(* CODESYS project OPAK_RFID.LIBRARY
   DefaultNamespace: ELA_OPAK_RFID
   Author: elrest Automationssysteme GmbH
   Title: OPAK_RFID
   DocFormat: reStructuredText
   Version: 3.5.0.0
   Description: Library to acces the RFID reader/writer on the EMC500 HW
   LanguageModelAttribute: qualified-access-only
   Company: elrest Automationssysteme GmbH

Project tree, tasks and I/O mapping:
  libraries: CAA Types Extern, * (CAA Technical Workgroup); CAA Behaviour Model, * (CAA Technical Workgroup); CAA FB Factory, * (CAA Technical Workgroup)
  00000000-0000-0000-0000-000000000000|D:\CoDeSys\LibrariesV3\trunk\Intern\CAA\CAA Template\3.2.0.3 draft\Prefix.pdf
  00000000-0000-0000-0000-000000000000|D:\CoDeSys\LibrariesV3\trunk\Intern\CAA\CAA Template\3.4.0.0 draft\Placeholder.xml
  00000000-0000-0000-0000-000000000000|D:\CoDeSys\LibrariesV3\trunk\Intern\CAA\CAA Template\3.5.2.0 draft\Placeholder.xml
  Libname/
    Enums/
      data type ERROR
    Function Blocks/
    Functions/
      function isTagPresent [ST]
      function getTagID [ST]
      function readFromTag [ST]
      function writeToTag [ST]
    GlobalConstants/
      global variables Constants
    GlobalVariables/
      global variables Variables
    Interfaces/
    Structs/
    Templates/
      Behaviour Model/
        function block ETrigA_Temp [ST]: prvAbort, prvCyclicAction, prvResetOutputs, prvStart
        function block ETrigTlA_Temp [ST]: prvAbort, prvCyclicAction, prvResetOutputs, prvStart
        function block ETrigTl_Temp [ST]: prvAbort, prvCyclicAction, prvResetOutputs, prvStart
        function block ETrigToA_Temp [ST]: prvAbort, prvCyclicAction, prvResetOutputs, prvStart
        function block ETrigToTlA_Temp [ST]: prvAbort, prvCyclicAction, prvResetOutputs, prvStart
        function block ETrigToTl_Temp [ST]: prvAbort, prvCyclicAction, prvResetOutputs, prvStart
        function block ETrigTo_Temp [ST]: prvAbort, prvCyclicAction, prvResetOutputs, prvStart
        function block ETrig_Temp [ST]: prvAbort, prvCyclicAction, prvResetOutputs, prvStart
        function block LTrig_Temp [ST]: prvAbort, prvCyclicAction, prvResetOutputs, prvStart
      FB Factory/
        function block CustomData [ST]
        function block CustomFB [ST]: prvInstInit
        function block CustomFBFactory_heap [ST]: Create, prvInstCount, prvInstPoolExtendsFactor, prvInstSize
        function block CustomFBFactory_static [ST]: Create, prvInstPoolAdr, prvInstPoolSize, prvInstSize
    Types/
  Projektinformationen/
    function GetCompany [ST]
    function GetTitle [ST]
    function GetVersion [ST]
    function GetTextProperty [ST]
    function GetNumberProperty [ST]
    function GetBooleanProperty [ST]
    function GetVersionProperty [ST]
*)

// Libname/Enums/ERROR
{attribute 'qualified_only'}
//{attribute 'conditionalshow'}
//{attribute 'conditionalshow' := 'SomeText'}
//{attribute 'hide'}
TYPE ERROR : (NO_ERROR, TIME_OUT); END_TYPE

// Libname/GlobalConstants/Constants
{attribute 'qualified_only'}
//{attribute 'conditionalshow'}
//{attribute 'conditionalshow' := 'SomeText'}
//{attribute 'hide'}
VAR_GLOBAL CONSTANT
	gc_iDummy : INT := 42; /// This is a dummy global constant variable
END_VAR

// Libname/GlobalVariables/Variables
{attribute 'qualified_only'}
//{attribute 'conditionalshow'}
//{attribute 'conditionalshow' := 'SomeText'}
//{attribute 'hide'}
VAR_GLOBAL
	g_iDummy : INT; /// This is a dummy global variable
END_VAR

// Libname/Templates/Behaviour Model/ETrigA_Temp
//{attribute 'hide_all_locals'}
//{attribute 'conditionalshow_all_locals' := 'SomeText'}
//{attribute 'conditionalshow_all_locals'}
//{attribute 'conditionalshow' := 'SomeText'}
//{attribute 'conditionalshow'}
//{attribute 'hide'}
FUNCTION_BLOCK ETrigA_Temp EXTENDS CBM.ETrigA
VAR_INPUT
	(* specific Inputs *)
END_VAR
VAR_OUTPUT
	eError : ERROR;
	(* specific Outputs *)
END_VAR
VAR
	(* specific vars *)
END_VAR

SUPER^();
IF iError = CBM.ERROR.TIME_OUT THEN
	eError := ERROR.TIME_OUT;
ELSE
	eError := iError;
END_IF

{attribute 'hide'}
METHOD prvAbort : BOOL
VAR_INPUT
END_VAR
VAR
END_VAR
IF xError THEN (* abort because of error *)
	(* TODO: insert specific Code here *)
ELSE (* user abort *)
	(* TODO: insert specific Code here *)
END_IF
xAbortInProgress:= FALSE;
END_METHOD

{attribute 'hide'}
METHOD prvCyclicAction : BOOL
VAR_INPUT
END_VAR
VAR
END_VAR
(* TODO: insert specific Code here *)
xDone:= TRUE;
(* if an error occurs, set iError to a value else than zero instead of xDone:= TRUE *)
(* to keep repeat loop *)
END_METHOD

{attribute 'hide'}
METHOD prvResetOutputs : BOOL
VAR_INPUT
END_VAR
VAR
END_VAR
(* TODO: insert specific Code here *)
SUPER^.prvResetOutputs();
END_METHOD

{attribute 'hide'}
METHOD prvStart : BOOL
VAR_INPUT
END_VAR
VAR
END_VAR
(* this code is called, when the application is started (rising edge of xExecute *)
(* TODO: copy specific input variables into local copies *)
(* TODO: insert specific Code here *)
;
END_METHOD

END_FUNCTION_BLOCK

// Libname/Templates/Behaviour Model/ETrigTlA_Temp
//{attribute 'hide_all_locals'}
//{attribute 'conditionalshow_all_locals' := 'SomeText'}
//{attribute 'conditionalshow_all_locals'}
//{attribute 'conditionalshow' := 'SomeText'}
//{attribute 'conditionalshow'}
//{attribute 'hide'}
FUNCTION_BLOCK ETrigTlA_Temp EXTENDS CBM.ETrigTlA
VAR_INPUT
	(* specific Inputs *)
END_VAR
VAR_OUTPUT
	eError : ERROR;
	(* specific Outputs *)
END_VAR
VAR
	(* specific vars *)
END_VAR

SUPER^();
IF iError = CBM.ERROR.TIME_OUT THEN
	eError := ERROR.TIME_OUT;
ELSE
	eError := iError;
END_IF

{attribute 'hide'}
METHOD prvAbort : BOOL
VAR_INPUT
END_VAR
VAR
END_VAR
IF xError THEN (* abort because of error *)
	(* TODO: insert specific Code here *)
ELSE (* user abort *)
	(* TODO: insert specific Code here *)
END_IF
xAbortInProgress:= FALSE;
END_METHOD

{attribute 'hide'}
METHOD prvCyclicAction : BOOL
VAR_INPUT
END_VAR
VAR
END_VAR
(* TODO: insert specific Code here *)
xDone:= TRUE;
(* if an error occurs, set iError to a value else than zero instead of xDone:= TRUE *)
(* to keep repeat loop *)
END_METHOD

{attribute 'hide'}
METHOD prvResetOutputs : BOOL
VAR_INPUT
END_VAR
VAR
END_VAR
(* TODO: insert specific Code here *)
SUPER^.prvResetOutputs();
END_METHOD

{attribute 'hide'}
METHOD prvStart : BOOL
VAR_INPUT
END_VAR
VAR
END_VAR
(* this code is called, when the application is started (rising edge of xExecute *)
(* TODO: copy specific input variables into local copies *)
(* TODO: insert specific Code here *)
;
END_METHOD

END_FUNCTION_BLOCK

// Libname/Templates/Behaviour Model/ETrigTl_Temp
//{attribute 'hide_all_locals'}
//{attribute 'conditionalshow_all_locals' := 'SomeText'}
//{attribute 'conditionalshow_all_locals'}
//{attribute 'conditionalshow' := 'SomeText'}
//{attribute 'conditionalshow'}
//{attribute 'hide'}
FUNCTION_BLOCK ETrigA_Temp EXTENDS CBM.ETrigTl
VAR_INPUT
	(* specific Inputs *)
END_VAR
VAR_OUTPUT
	eError : ERROR;
	(* specific Outputs *)
END_VAR
VAR
	(* specific vars *)
END_VAR

SUPER^();
IF iError = CBM.ERROR.TIME_OUT THEN
	eError := ERROR.TIME_OUT;
ELSE
	eError := iError;
END_IF

{attribute 'hide'}
METHOD prvAbort : BOOL
VAR_INPUT
END_VAR
VAR
END_VAR
IF xError THEN (* abort because of error *)
	(* TODO: insert specific Code here *)
ELSE (* user abort *)
	(* TODO: insert specific Code here *)
END_IF
xAbortInProgress:= FALSE;
END_METHOD

{attribute 'hide'}
METHOD prvCyclicAction : BOOL
VAR_INPUT
END_VAR
VAR
END_VAR
(* TODO: insert specific Code here *)
xDone:= TRUE;
(* if an error occurs, set iError to a value else than zero instead of xDone:= TRUE *)
(* to keep repeat loop *)
END_METHOD

{attribute 'hide'}
METHOD prvResetOutputs : BOOL
VAR_INPUT
END_VAR
VAR
END_VAR
(* TODO: insert specific Code here *)
SUPER^.prvResetOutputs();
END_METHOD

{attribute 'hide'}
METHOD prvStart : BOOL
VAR_INPUT
END_VAR
VAR
END_VAR
(* this code is called, when the application is started (rising edge of xExecute *)
(* TODO: copy specific input variables into local copies *)
(* TODO: insert specific Code here *)
;
END_METHOD

END_FUNCTION_BLOCK

// Libname/Templates/Behaviour Model/ETrigToA_Temp
//{attribute 'hide_all_locals'}
//{attribute 'conditionalshow_all_locals' := 'SomeText'}
//{attribute 'conditionalshow_all_locals'}
//{attribute 'conditionalshow' := 'SomeText'}
//{attribute 'conditionalshow'}
//{attribute 'hide'}
FUNCTION_BLOCK ETrigToA_Temp EXTENDS CBM.ETrigToA
VAR_INPUT
	(* specific Inputs *)
END_VAR
VAR_OUTPUT
	eError : ERROR;
	(* specific Outputs *)
END_VAR
VAR
	(* specific vars *)
END_VAR

SUPER^();
IF iError = CBM.ERROR.TIME_OUT THEN
	eError := ERROR.TIME_OUT;
ELSE
	eError := iError;
END_IF

{attribute 'hide'}
METHOD prvAbort : BOOL
VAR_INPUT
END_VAR
VAR
END_VAR
IF xError THEN (* abort because of error *)
	(* TODO: insert specific Code here *)
ELSE (* user abort *)
	(* TODO: insert specific Code here *)
END_IF
xAbortInProgress:= FALSE;
END_METHOD

{attribute 'hide'}
METHOD prvCyclicAction : BOOL
VAR_INPUT
END_VAR
VAR
END_VAR
(* TODO: insert specific Code here *)
xDone:= TRUE;
(* if an error occurs, set iError to a value else than zero instead of xDone:= TRUE *)
END_METHOD

{attribute 'hide'}
METHOD prvResetOutputs : BOOL
VAR_INPUT
END_VAR
VAR
END_VAR
(* TODO: insert specific Code here *)
SUPER^.prvResetOutputs();
END_METHOD

{attribute 'hide'}
METHOD prvStart : BOOL
VAR_INPUT
END_VAR
VAR
END_VAR
(* this code is called, when the application is started (rising edge of xExecute *)
(* TODO: copy specific input variables into local copies *)
(* TODO: insert specific Code here *)
;
END_METHOD

END_FUNCTION_BLOCK

// Libname/Templates/Behaviour Model/ETrigToTlA_Temp
//{attribute 'hide_all_locals'}
//{attribute 'conditionalshow_all_locals' := 'SomeText'}
//{attribute 'conditionalshow_all_locals'}
//{attribute 'conditionalshow' := 'SomeText'}
//{attribute 'conditionalshow'}
//{attribute 'hide'}
FUNCTION_BLOCK ETrigToTlA_Temp EXTENDS CBM.ETrigToTlA
VAR_INPUT
	(* specific Inputs *)
END_VAR
VAR_OUTPUT
	eError : ERROR;
	(* specific Outputs *)
END_VAR
VAR
	(* specific vars *)
END_VAR

SUPER^();
IF iError = CBM.ERROR.TIME_OUT THEN
	eError := ERROR.TIME_OUT;
ELSE
	eError := iError;
END_IF

{attribute 'hide'}
METHOD prvAbort : BOOL
VAR_INPUT
END_VAR
VAR
END_VAR
IF xError THEN (* abort because of error *)
	(* TODO: insert specific Code here *)
ELSE (* user abort *)
	(* TODO: insert specific Code here *)
END_IF
xAbortInProgress:= FALSE;
END_METHOD

{attribute 'hide'}
METHOD prvCyclicAction : BOOL
VAR_INPUT
END_VAR
VAR
END_VAR
(* TODO: insert specific Code here *)
xDone:= TRUE;
(* if an error occurs, set iError to a value else than zero instead of xDone:= TRUE *)
(* to keep repeat loop *)
END_METHOD

{attribute 'hide'}
METHOD prvResetOutputs : BOOL
VAR_INPUT
END_VAR
VAR
END_VAR
(* TODO: insert specific Code here *)
SUPER^.prvResetOutputs();
END_METHOD

{attribute 'hide'}
METHOD prvStart : BOOL
VAR_INPUT
END_VAR
VAR
END_VAR
(* this code is called, when the application is started (rising edge of xExecute *)
(* TODO: copy specific input variables into local copies *)
(* TODO: insert specific Code here *)
;
END_METHOD

END_FUNCTION_BLOCK

// Libname/Templates/Behaviour Model/ETrigToTl_Temp
//{attribute 'hide_all_locals'}
//{attribute 'conditionalshow_all_locals' := 'SomeText'}
//{attribute 'conditionalshow_all_locals'}
//{attribute 'conditionalshow' := 'SomeText'}
//{attribute 'conditionalshow'}
//{attribute 'hide'}
FUNCTION_BLOCK ETrigToTl_Temp EXTENDS CBM.ETrigToTl
VAR_INPUT
	(* specific Inputs *)
END_VAR
VAR_OUTPUT
	eError : ERROR;
	(* specific Outputs *)
END_VAR
VAR
	(* specific vars *)
END_VAR

SUPER^();
IF iError = CBM.ERROR.TIME_OUT THEN
	eError := ERROR.TIME_OUT;
ELSE
	eError := iError;
END_IF

{attribute 'hide'}
METHOD prvAbort : BOOL
VAR_INPUT
END_VAR
VAR
END_VAR
IF xError THEN (* abort because of error *)
	(* TODO: insert specific Code here *)
ELSE (* user abort *)
	(* TODO: insert specific Code here *)
END_IF
xAbortInProgress:= FALSE;
END_METHOD

{attribute 'hide'}
METHOD prvCyclicAction : BOOL
VAR_INPUT
END_VAR
VAR
END_VAR
(* TODO: insert specific Code here *)
xDone:= TRUE;
(* if an error occurs, set iError to a value else than zero instead of xDone:= TRUE *)
(* to keep repeat loop *)
END_METHOD

{attribute 'hide'}
METHOD prvResetOutputs : BOOL
VAR_INPUT
END_VAR
VAR
END_VAR
(* TODO: insert specific Code here *)
SUPER^.prvResetOutputs();
END_METHOD

{attribute 'hide'}
METHOD prvStart : BOOL
VAR_INPUT
END_VAR
VAR
END_VAR
(* this code is called, when the application is started (rising edge of xExecute *)
(* TODO: copy specific input variables into local copies *)
(* TODO: insert specific Code here *)
;
END_METHOD

END_FUNCTION_BLOCK

// Libname/Templates/Behaviour Model/ETrigTo_Temp
//{attribute 'hide_all_locals'}
//{attribute 'conditionalshow_all_locals' := 'SomeText'}
//{attribute 'conditionalshow_all_locals'}
//{attribute 'conditionalshow' := 'SomeText'}
//{attribute 'conditionalshow'}
//{attribute 'hide'}
FUNCTION_BLOCK ETrigTo_Temp EXTENDS CBM.ETrigTo
VAR_INPUT
	(* specific Inputs *)
END_VAR
VAR_OUTPUT
	eError : ERROR;
	(* specific Outputs *)
END_VAR
VAR
	(* specific vars *)
END_VAR

SUPER^();
IF iError = CBM.ERROR.TIME_OUT THEN
	eError := ERROR.TIME_OUT;
ELSE
	eError := iError;
END_IF

{attribute 'hide'}
METHOD prvAbort : BOOL
VAR_INPUT
END_VAR
VAR
END_VAR
IF xError THEN (* abort because of error *)
	(* TODO: insert specific Code here *)
ELSE (* user abort *)
	(* TODO: insert specific Code here *)
END_IF
xAbortInProgress:= FALSE;
END_METHOD

{attribute 'hide'}
METHOD prvCyclicAction : BOOL
VAR_INPUT
END_VAR
VAR
END_VAR
(* TODO: insert specific Code here *)
xDone:= TRUE;
(* if an error occurs, set iError to a value else than zero instead of xDone:= TRUE *)
(* to keep repeat loop *)
END_METHOD

{attribute 'hide'}
METHOD prvResetOutputs : BOOL
VAR_INPUT
END_VAR
VAR
END_VAR
(* TODO: insert specific Code here *)
SUPER^.prvResetOutputs();
END_METHOD

{attribute 'hide'}
METHOD prvStart : BOOL
VAR_INPUT
END_VAR
VAR
END_VAR
(* this code is called, when the application is started (rising edge of xExecute *)
(* TODO: copy specific input variables into local copies *)
(* TODO: insert specific Code here *)
;
END_METHOD

END_FUNCTION_BLOCK

// Libname/Templates/Behaviour Model/ETrig_Temp
//{attribute 'hide_all_locals'}
//{attribute 'conditionalshow_all_locals' := 'SomeText'}
//{attribute 'conditionalshow_all_locals'}
//{attribute 'conditionalshow' := 'SomeText'}
//{attribute 'conditionalshow'}
//{attribute 'hide'}
FUNCTION_BLOCK ETrig_Temp EXTENDS CBM.ETrig
VAR_INPUT
	(* specific Inputs *)
END_VAR
VAR_OUTPUT
	eError : ERROR;
	(* specific Outputs *)
END_VAR
VAR
	(* specific vars *)
END_VAR

SUPER^();
IF iError = CBM.ERROR.TIME_OUT THEN
	eError := ERROR.TIME_OUT;
ELSE
	eError := iError;
END_IF

{attribute 'hide'}
METHOD prvAbort : BOOL
VAR_INPUT
END_VAR
VAR
END_VAR
IF xError THEN (* abort because of error *)
	(* TODO: insert specific Code here *)
ELSE (* user abort *)
	(* TODO: insert specific Code here *)
END_IF
xAbortInProgress:= FALSE;
END_METHOD

{attribute 'hide'}
METHOD prvCyclicAction : BOOL
VAR_INPUT
END_VAR
VAR
END_VAR
(* TODO: insert specific Code here *)
xDone:= TRUE;
(* if an error occurs, set iError to a value else than zero instead of xDone:= TRUE *)
(* to keep repeat loop *)
END_METHOD

{attribute 'hide'}
METHOD prvResetOutputs : BOOL
VAR_INPUT
END_VAR
VAR
END_VAR
(* TODO: insert specific Code here *)
SUPER^.prvResetOutputs();
END_METHOD

{attribute 'hide'}
METHOD prvStart : BOOL
VAR_INPUT
END_VAR
VAR
END_VAR
(* this code is called, when the application is started (rising edge of xExecute *)
(* TODO: copy specific input variables into local copies *)
(* TODO: insert specific Code here *)
;
END_METHOD

END_FUNCTION_BLOCK

// Libname/Templates/Behaviour Model/LTrig_Temp
//{attribute 'hide_all_locals'}
//{attribute 'conditionalshow_all_locals' := 'SomeText'}
//{attribute 'conditionalshow_all_locals'}
//{attribute 'conditionalshow' := 'SomeText'}
//{attribute 'conditionalshow'}
//{attribute 'hide'}
FUNCTION_BLOCK LTrig_Temp EXTENDS CBM.LTrig
VAR_INPUT
	(* specific Inputs *)
END_VAR
VAR_OUTPUT
	eError : ERROR;
	(* specific Outputs *)
END_VAR
VAR
	(* specific vars *)
END_VAR

SUPER^();
IF iError = CBM.ERROR.TIME_OUT THEN
	eError := ERROR.TIME_OUT;
ELSE
	eError := iError;
END_IF

{attribute 'hide'}
METHOD prvAbort : BOOL
VAR_INPUT
END_VAR
VAR
END_VAR
IF xError THEN (* abort because of error *)
	(* TODO: insert specific Code here *)
ELSE (* user abort *)
	(* TODO: insert specific Code here *)
END_IF
xAbortInProgress:= FALSE;
END_METHOD

{attribute 'hide'}
METHOD prvCyclicAction : BOOL
VAR_INPUT
END_VAR
VAR
END_VAR
(* TODO: insert specific Code here *)
xDone:= TRUE;
(* if an error occurs, set iError to a value else than zero instead of xDone:= TRUE *)
(* to keep repeat loop *)
END_METHOD

{attribute 'hide'}
METHOD prvResetOutputs : BOOL
VAR_INPUT
END_VAR
VAR
END_VAR
(* TODO: insert specific Code here *)
SUPER^.prvResetOutputs();
END_METHOD

{attribute 'hide'}
METHOD prvStart : BOOL
VAR_INPUT
END_VAR
VAR
END_VAR
(* this code is called, when the application is started (rising edge of xExecute *)
(* TODO: copy specific input variables into local copies *)
(* TODO: insert specific Code here *)
;
END_METHOD

END_FUNCTION_BLOCK

// Libname/Templates/FB Factory/CustomData
// This is a container to carry init data from the Create methode of the factory
// to the prvInstInit methode of the new generated function block instance
{attribute 'enable_dynamic_creation'}
//{attribute 'hide_all_locals'}
//{attribute 'conditionalshow_all_locals' := 'SomeText'}
//{attribute 'conditionalshow_all_locals'}
//{attribute 'conditionalshow' := 'SomeText'}
//{attribute 'conditionalshow'}
//{attribute 'hide'}
FUNCTION_BLOCK CustomData EXTENDS FBF.InstanceData
VAR_INPUT
	(* Todo: Add your application specific data as input variables *)
END_VAR

(* !! Do not add any executable code here !! *)
SUPER^();

END_FUNCTION_BLOCK

// Libname/Templates/FB Factory/CustomFB
{attribute 'enable_dynamic_creation'}
//{attribute 'hide_all_locals'}
//{attribute 'conditionalshow_all_locals' := 'SomeText'}
//{attribute 'conditionalshow_all_locals'}
//{attribute 'conditionalshow' := 'SomeText'}
//{attribute 'conditionalshow'}
//{attribute 'hide'}
FUNCTION_BLOCK CustomFB EXTENDS FBF.InstanceBase;
VAR_INPUT
END_VAR
VAR_OUTPUT
END_VAR
VAR
END_VAR

SUPER^();

// This methode is called from the factory to give a chance
// to initialize the new fb instance with the content of itfData
//{attribute 'hide_all_locals'}
//{attribute 'conditionalshow_all_locals' := 'SomeText'}
//{attribute 'conditionalshow_all_locals'}
//{attribute 'conditionalshow' := 'SomeText'}
//{attribute 'conditionalshow'}
//{attribute 'hide'}
METHOD prvInstInit : FBF.ERROR
VAR_INPUT
	itfData : IData; 
END_VAR
VAR
	pData : POINTER TO CustomData;
	xOk : BOOL;
END_VAR
SUPER^.prvInstInit(itfData);
xOk := __QUERYPOINTER(itfData, pData);
IF xOk THEN
	(* THIS^.iLocalVar := pData^.iInitValue *);
END_IF
END_METHOD

END_FUNCTION_BLOCK

// Libname/Templates/FB Factory/CustomFBFactory_heap
// This is a template for a factory with an heap based extendable memory pool
{attribute 'enable_dynamic_creation'}
//{attribute 'hide_all_locals'}
//{attribute 'conditionalshow_all_locals' := 'SomeText'}
//{attribute 'conditionalshow_all_locals'}
//{attribute 'conditionalshow' := 'SomeText'}
//{attribute 'conditionalshow'}
//{attribute 'hide'}
FUNCTION_BLOCK CustomFBFactory_heap EXTENDS FactoryBase
VAR
END_VAR

SUPER^();

(* Please replace CustonFB with your specific function block type *)
(* There is no need to change anything else !!! *)
METHOD Create : POINTER TO CustomFB
VAR_INPUT
	itfData : FBF.IData;
END_VAR
VAR_OUTPUT
	eError : FBF.ERROR;
END_VAR
VAR
	hInst : CAA.HANDLE;
	itfInst : FBF.IInstance;
	xOk : BOOL;
END_VAR
(* !!! This code must not be subject to change !!! *)
hInst := SUPER^.prvAllocInstMem(eError => eError);
Create := SUPER^.prvGetInstPointer(hInst);
IF Create <> 0 AND eError = FBF.ERROR.NO_ERROR THEN

	{implicit on}
	Create^.__vfInit();
	Create^.FB_Init(TRUE, FALSE);
	{implicit off}

	xOk := __QUERYINTERFACE(Create^, itfInst);
	IF xOk THEN
		xOk := SUPER^.prvInstInit(itfInst, hInst, itfData, eError=>eError);
	ELSE
		eError := FBF.ERROR.WRONG_INTERFACE;
	END_IF

	IF NOT xOk THEN
		SUPER^.prvFreeInstMem(hInst);
		Create := CAA.gc_pNULL;
	END_IF
END_IF
END_METHOD

//{attribute 'conditionalshow' := 'SomeText'}
//{attribute 'conditionalshow'}
//{attribute 'hide'}
PROPERTY prvInstCount : CAA.COUNT (* ctInst *)
GET
(* Please choose a proper value for prvInstCount *)
prvInstCount := 10;
END_GET
END_PROPERTY

//{attribute 'conditionalshow' := 'SomeText'}
//{attribute 'conditionalshow'}
//{attribute 'hide'}
PROPERTY prvInstPoolExtendsFactor : USINT (* usiFactor [0..x%] *)
GET
(* Please choose a proper value for prvInstPoolExtendsFactor *)
(* This value will be interpreted as a 0..x% size extendsion related to the original size of the pool *)
prvInstPoolExtendsFactor := 20;
END_GET
END_PROPERTY

//{attribute 'conditionalshow' := 'SomeText'}
//{attribute 'conditionalshow'}
//{attribute 'hide'}
PROPERTY prvInstSize : CAA.SIZE (* szInst *)
GET
(* Please replace CustomFB with your specific function block type *)
prvInstSize := sizeof(CustomFB);
END_GET
END_PROPERTY

END_FUNCTION_BLOCK

// Libname/Templates/FB Factory/CustomFBFactory_static
// This is a template for a factory with an static iec memory based memory pool which a fixed capacity
{attribute 'enable_dynamic_creation'}
//{attribute 'hide_all_locals'}
//{attribute 'conditionalshow_all_locals' := 'SomeText'}
//{attribute 'conditionalshow_all_locals'}
//{attribute 'conditionalshow' := 'SomeText'}
//{attribute 'conditionalshow'}
//{attribute 'hide'}
FUNCTION_BLOCK CustomFBFactory_static EXTENDS FactoryBase
VAR
	// Please change the size of abyPoolMemory with your specific application need
	abyPoolMemory : ARRAY[0..529] OF BYTE;
END_VAR

SUPER^();

(* Please replace CustonFB with our specific function block type *)
(* There is no need to change anything else !!! *)
METHOD Create : POINTER TO CustomFB
VAR_INPUT
	itfData : FBF.IData;
END_VAR
VAR_OUTPUT
	eError : FBF.ERROR;
END_VAR
VAR
	hInst : CAA.HANDLE;
	itfInst : FBF.IInstance;
	xOk : BOOL;
END_VAR
(* !!! This code must not be subject to change !!! *)
hInst := SUPER^.prvAllocInstMem(eError => eError);
Create := SUPER^.prvGetInstPointer(hInst);
IF Create <> 0 AND eError = FBF.ERROR.NO_ERROR THEN

	{implicit on}
	Create^.__vfInit();
	Create^.FB_Init(TRUE, FALSE);
	{implicit off}

	xOk := __QUERYINTERFACE(Create^, itfInst);
	IF xOk THEN
		xOk := SUPER^.prvInstInit(itfInst, hInst, itfData, eError=>eError);
	ELSE
		eError := FBF.ERROR.WRONG_INTERFACE;
	END_IF

	IF NOT xOk THEN
		SUPER^.prvFreeInstMem(hInst);
		Create := CAA.gc_pNULL;
	END_IF
END_IF
END_METHOD

//{attribute 'conditionalshow' := 'SomeText'}
//{attribute 'conditionalshow'}
//{attribute 'hide'}
PROPERTY prvInstPoolAdr : CAA.PVOID (* pPool *)
GET
prvInstPoolAdr := ADR(abyPoolMemory);
END_GET
END_PROPERTY

//{attribute 'conditionalshow' := 'SomeText'}
//{attribute 'conditionalshow'}
//{attribute 'hide'}
PROPERTY prvInstPoolSize : CAA.SIZE (* szPool *)
GET
prvInstPoolSize := sizeof(abyPoolMemory);
END_GET
END_PROPERTY

//{attribute 'conditionalshow' := 'SomeText'}
//{attribute 'conditionalshow'}
//{attribute 'hide'}
PROPERTY prvInstSize : CAA.SIZE (* szInst *)
GET
(* Please replace CustomFB with your specific function block type *)
prvInstSize := sizeof(CustomFB);
END_GET
END_PROPERTY

END_FUNCTION_BLOCK

// Libname/Functions/isTagPresent
FUNCTION isTagPresent : BOOL (* Returns true if a Tag was detected with RFID*)
VAR_INPUT
END_VAR
VAR
END_VAR

END_FUNCTION

// Libname/Functions/getTagID
FUNCTION getTagID : STRING (* Returns Tag's serial number if present *)
VAR_INPUT
END_VAR
VAR
END_VAR

END_FUNCTION

// Libname/Functions/readFromTag
FUNCTION readFromTag : UINT (*Number of bytes read, 0 if no TAG present*) (*At the moment only fixed 4 bytes can be read from device, needs fix*)
VAR_INPUT
	addr : UINT; (* First byte to read from *)
	len : UINT; (* Number of Bytes to read *)
	buf : POINTER TO DWORD; (* Pointer to a buffer, must have at least len size *)
END_VAR
VAR
END_VAR

END_FUNCTION

// Libname/Functions/writeToTag
FUNCTION writeToTag : UINT (*Returns number of bytes written *)
VAR_INPUT
	addr : UINT; (* First byte to read from *)
	len : UINT; (* Number of Bytes to read *)
	buf : POINTER TO BYTE; (* Pointer to a buffer, must have at least len size *)
END_VAR
VAR
END_VAR

END_FUNCTION

// Projektinformationen/GetCompany
// This function has been automatically generated from the project information.
{attribute 'signature_flag' := '1073741824'}
{attribute 'register_in_runtime'}
FUNCTION GetCompany : WSTRING
VAR_INPUT
	
END_VAR

GetCompany := "elrest Automationssysteme GmbH";

END_FUNCTION

// Projektinformationen/GetTitle
// This function has been automatically generated from the project information.
{attribute 'signature_flag' := '1073741824'}
{attribute 'register_in_runtime'}
FUNCTION GetTitle : WSTRING
VAR_INPUT
	
END_VAR

GetTitle := "OPAK_RFID";

END_FUNCTION

// Projektinformationen/GetVersion
// This function has been automatically generated from the project information.
{attribute 'signature_flag' := '1073741824'}
{attribute 'register_in_runtime'}
FUNCTION GetVersion : VERSION
VAR_INPUT
	
END_VAR

GetVersion.uiMajor := 3;
GetVersion.uiMinor := 5;
GetVersion.uiServicePack := 0;
GetVersion.uiPatch := 0;

END_FUNCTION

// Projektinformationen/GetTextProperty
// This function has been automatically generated from the project information.
{attribute 'signature_flag' := '1073741824'}
{attribute 'register_in_runtime'}
FUNCTION GetTextProperty : WSTRING
VAR_INPUT
	stKey: WSTRING;
END_VAR

IF stKey = "Author" THEN
	GetTextProperty := "elrest Automationssysteme GmbH";
ELSIF stKey = "Company" THEN
	GetTextProperty := "elrest Automationssysteme GmbH";
ELSIF stKey = "DefaultNamespace" THEN
	GetTextProperty := "ELA_OPAK_RFID";
ELSIF stKey = "Description" THEN
	GetTextProperty := "Library to acces the RFID reader/writer on the EMC500 HW";
ELSIF stKey = "DocFormat" THEN
	GetTextProperty := "reStructuredText";
ELSIF stKey = "LanguageModelAttribute" THEN
	GetTextProperty := "qualified-access-only";
ELSIF stKey = "Project" THEN
	GetTextProperty := "LibOPAK_RFID";
ELSIF stKey = "Title" THEN
	GetTextProperty := "OPAK_RFID";
ELSE
	GetTextProperty := "";
END_IF

END_FUNCTION

// Projektinformationen/GetNumberProperty
// This function has been automatically generated from the project information.
{attribute 'signature_flag' := '1073741824'}
{attribute 'register_in_runtime'}
FUNCTION GetNumberProperty : DINT
VAR_INPUT
	stKey: WSTRING;
END_VAR

GetNumberProperty := 0;

END_FUNCTION

// Projektinformationen/GetBooleanProperty
// This function has been automatically generated from the project information.
{attribute 'signature_flag' := '1073741824'}
{attribute 'register_in_runtime'}
FUNCTION GetBooleanProperty : BOOL
VAR_INPUT
	stKey: WSTRING;
END_VAR

IF stKey = "IsEndUserLibrary" THEN
	GetBooleanProperty := FALSE;
ELSIF stKey = "Released" THEN
	GetBooleanProperty := FALSE;
ELSE
	GetBooleanProperty := FALSE;
END_IF

END_FUNCTION

// Projektinformationen/GetVersionProperty
// This function has been automatically generated from the project information.
{attribute 'signature_flag' := '1073741824'}
{attribute 'register_in_runtime'}
FUNCTION GetVersionProperty : VERSION
VAR_INPUT
	stKey: WSTRING;
END_VAR

IF stKey = "Version" THEN
	GetVersionProperty.uiMajor := 3;
	GetVersionProperty.uiMinor := 5;
	GetVersionProperty.uiServicePack := 0;
	GetVersionProperty.uiPatch := 0;
ELSE
	GetVersionProperty.uiMajor := 0;
	GetVersionProperty.uiMinor := 0;
	GetVersionProperty.uiServicePack := 0;
	GetVersionProperty.uiPatch := 0;
END_IF

END_FUNCTION
